INTERFACE ITF_Actuator EXTENDS ITF_BaseControlElement

METHOD IsEnd : BOOL
VAR_INPUT
END_VAR
END_METHOD

METHOD PUBLIC IsStart : BOOL
VAR_INPUT
END_VAR
END_METHOD

(*			
	EVERDE sp. z o.o.
	Rafał Osajda		31.03.2025		TC 4024.66
	Uruchomienie cyklu przesuwania do początku
*)
METHOD PUBLIC MoveToEnd
VAR_INPUT
END_VAR
END_METHOD

(*			
	EVERDE sp. z o.o.
	Rafał Osajda		31.03.2025		TC 4024.66
	Uruchomienie cyklu przesuwania do początku
*)
METHOD PUBLIC MoveToStart
VAR_INPUT
END_VAR
END_METHOD

METHOD PUBLIC MovingToEndBusy : BOOL
VAR_INPUT
END_VAR
END_METHOD

METHOD PUBLIC MovingToEndFirstCycyle : BOOL
VAR_INPUT
END_VAR
END_METHOD

METHOD PUBLIC MovingToEndStatus : BOOL
VAR_INPUT
END_VAR
END_METHOD

METHOD PUBLIC MovingToStartBusy : BOOL
VAR_INPUT
END_VAR
END_METHOD

METHOD PUBLIC MovingToStartFirstCycle : BOOL
VAR_INPUT
END_VAR
END_METHOD

METHOD PUBLIC MovingToStartStatus : BOOL
VAR_INPUT
END_VAR
END_METHOD

END_INTERFACE

(* stored: Version 1.1.0.1
   Itf ITF_Actuator: Id {e06c23bd-6d65-496f-85d8-cbcf241671e7}
   Method IsEnd: Id {5cd55504-ae4a-0d73-14b7-4b484de38665}
   Method IsStart: Id {f633a98b-80df-0a9b-2eba-58e57903f185}
   Method MoveToEnd: Id {f6392d74-a86c-4303-977c-fdb5f4adf54b}
   Method MoveToStart: Id {fbf1076c-cb09-48ba-9d74-e16996404ec4}
   Method MovingToEndBusy: Id {6db5a6bb-6d3f-498b-9ec9-9eb7ac149e58}
   Method MovingToEndFirstCycyle: Id {8b4a7726-4dc8-4063-b1e9-5013e1c35c07}
   Method MovingToEndStatus: Id {10b0d999-7674-4b98-98c9-6425da0ab057}
   Method MovingToStartBusy: Id {8bab9372-1e44-4bc0-9cad-51ba9eff62a5}
   Method MovingToStartFirstCycle: Id {d1327414-71c9-43c3-beea-115acc1bdaae}
   Method MovingToStartStatus: Id {dada06ec-4aa4-4082-a473-d23b386c72ea} *)
